Universal Robots PolyScope program: 6-movel_with_relative_waypoint.urp

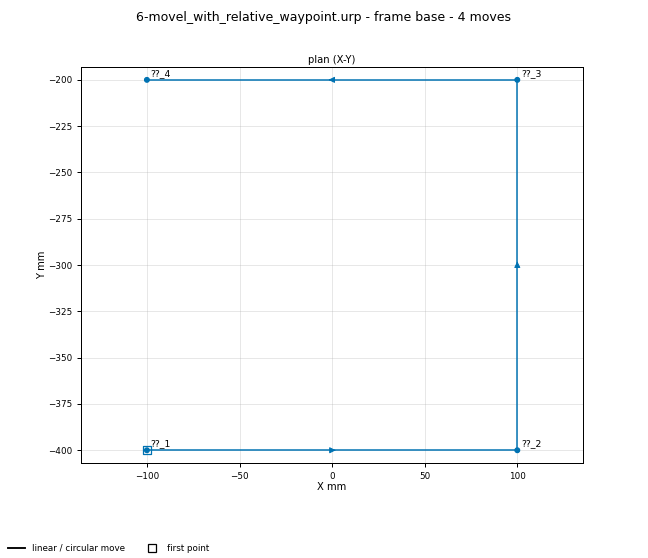
[picture p0: tool path of 6-movel_with_relative_waypoint.urp in frame base, 4 of 4 moves have a stored position in this frame; points joined in program order, loops and branches not executed]
ProgramRoot directory=/home/ur/ursim-3.1/programs/basic training/6-movel_with_relative_waypoint; kinematics=(a=[0, -0.425, -0.39225, 0, 0, 0], d=[0.08916, 0, 0, 0.10915, 0.09465, 0.0823], alpha=[1.5708, 0, 0, 1.5708, -1.5708, 0], deltaTheta=[0, 0, 0, 0, 0, 0], status=notInitialized); lastSavedInVersion=(project__name=Polyscope, major__version=3, minor__version=1, svn__revision=17195, build__date=Mar 11 2015, 13:02:28); name=6-movel_with_relative_waypoint; programVersion=(project__name=Polyscope, major__version=3, minor__version=1, svn__revision=17195, build__date=Mar 11 2015, 13:02:28); robotEnvironmentFileName=default; serialNumberRobot=2014350001
  MainProgram cartesianAcceleration=1.2; cartesianSpeed=0.25; jointAcceleration=1.3962634015954636; jointSpeed=1.0471975511965976; sharedProcessMoveBlendRadius=0.025; motionType=JOINT_SPACE
    Move cartesianAcceleration=1.2; cartesianSpeed=0.25; jointAcceleration=1.3962634015954636; jointSpeed=1.0471975511965976; sharedProcessMoveBlendRadius=0.025; motionType=CARTESIAN_SPACE
      Waypoint blendRadius=0.05; cartesianAcceleration=1.2; cartesianSpeed=0.25; jointAcceleration=1.3962634015954636; jointSpeed=1.0471975511965976; nextMotionTime=2.0; stoppoint=true; useSharedBlendParameter=true; useSharedParameters=true; outputFlangePose=(pos=(x=-0.10000000065989616, y=-0.40000000104212996, z=0.1999999982306596), rot=(x=-0.0012209830283997337, y=3.116276481240887, z=0.0388919161681283)); position=TCP in base x=-100 y=-400 z=200 mm, rx=-0.0012 ry=3.1163 rz=0.0389 rad; joints [-88.988, -88.3, -127.491, -55.614, 91.461, 0.95] deg; positionType=FIXED_POSITION; waypointPoseInFeatureCoordinates=(pos=(x=-0.09999996819589951, y=-0.40000005265404437, z=0.1999999632555712), rot=(x=-0.0012210995530369398, y=3.1162764787073427, z=0.0388923209577584)); name=路点_1
      Waypoint blendRadius=0.05; cartesianAcceleration=1.2; cartesianSpeed=0.25; jointAcceleration=1.3962634015954636; jointSpeed=1.0471975511965976; nextMotionTime=2.0; stoppoint=true; useSharedBlendParameter=true; useSharedParameters=true; outputFlangePose=(pos=(x=0.09999999955452232, y=-0.4000000526540431, z=0.20000000000000356), rot=(x=-0.0012210995519186247, y=3.1162764787073653, z=0.03889232095772719)); position=TCP in base x=100 y=-400 z=200 mm, rx=-0.0012 ry=3.1163 rz=0.0389 rad; joints [-61.016, -88.295, -127.75, -54.511, 91.949, 28.93] deg; positionType=RELATIVE_POSITION; waypointPoseInFeatureCoordinates=(pos=(x=0.09999998881554663, y=-0.4000000991077624, z=0.20000003628695473), rot=(x=-0.0012209612224475359, y=3.116276382769786, z=0.03889219223422068)); name=路点_2; relativeFromJointPositionVector=(joint=[-1.55313, -1.54113, -2.22514, -0.97064, 1.5963, 0.01657], isUndefined=false); relativeFromToolAxisAngle=(x=-0.0012210966507876907, y=3.1162764787312773, z=0.03889232099443211); relativeFromToolPosition=(x=-0.09999996819589951, y=-0.40000005265404437, z=0.1999999632555712)
      Waypoint blendRadius=0.05; cartesianAcceleration=1.2; cartesianSpeed=0.25; jointAcceleration=1.3962634015954636; jointSpeed=1.0471975511965976; nextMotionTime=2.0; stoppoint=true; useSharedBlendParameter=true; useSharedParameters=true; outputFlangePose=(pos=(x=0.09999998881558855, y=-0.20000000019511877, z=0.20000003628698113), rot=(x=-0.001220961222489403, y=3.116276382769804, z=0.03889219223416196)); position=TCP in base x=100 y=-200 z=200 mm, rx=-0.0012 ry=3.1163 rz=0.0389 rad; joints [-35.055, -51.443, -149.443, -68.76, 91.996, 54.906] deg; positionType=RELATIVE_POSITION; waypointPoseInFeatureCoordinates=(pos=(x=0.09999994119250635, y=-0.2000000164556638, z=0.20000002059083857), rot=(x=-0.0012206277928056932, y=3.116276456281894, z=0.03889217035544603)); name=路点_3; relativeFromJointPositionVector=(joint=[-1.06493, -1.54103, -2.22965, -0.9514, 1.60482, 0.50492], isUndefined=false); relativeFromToolAxisAngle=(x=-0.0012209612224476384, y=3.1162763827697897, z=0.03889219223422073); relativeFromToolPosition=(x=0.09999998881554663, y=-0.4000000991077624, z=0.20000003628695473)
      Waypoint blendRadius=0.05; cartesianAcceleration=1.2; cartesianSpeed=0.25; jointAcceleration=1.3962634015954636; jointSpeed=1.0471975511965976; nextMotionTime=2.0; stoppoint=true; useSharedBlendParameter=true; useSharedParameters=true; outputFlangePose=(pos=(x=-0.10000000051947, y=-0.20000001645565174, z=0.20000002059086222), rot=(x=-0.0012206277927958148, y=3.1162764562819243, z=0.03889217035537928)); position=TCP in base x=-100 y=-200 z=200 mm, rx=-0.0012 ry=3.1163 rz=0.0389 rad; joints [-87.972, -51.697, -148.925, -70.758, 91.486, 1.966] deg; positionType=RELATIVE_POSITION; waypointPoseInFeatureCoordinates=(pos=(x=-0.10000000149826872, y=-0.20000001703660555, z=0.20000009753562856), rot=(x=-0.0012206551156430997, y=3.116276500636825, z=0.038891741712667925)); name=路点_4; relativeFromJointPositionVector=(joint=[-0.61183, -0.89785, -2.60827, -1.20009, 1.60563, 0.95829], isUndefined=false); relativeFromToolAxisAngle=(x=-0.0012206277928057542, y=3.116276456281862, z=0.038892170355445635); relativeFromToolPosition=(x=0.09999994119250635, y=-0.2000000164556638, z=0.20000002059083857)
